FUNCTION proj1_TupleStruct_3: DINT
VAR_INPUT
    tuple: TupleStruct_3;
END_VAR

proj1_TupleStruct_3 := tuple.field1;

END_FUNCTION

(* stored: ProductVersion 3.1.0.18, Version 1.1.0.1 *)
